FUNCTION_BLOCK Q_ObjHideShow (* Command Hide/Show Object (Container) ( Part 6 - F.2 ) *)
  (* Standard: ISO 11783-6; Description: This command is used to change the value of an object. It applies only to objects that have a numeric value attribute. \retval      iso_s16 - #E_NO_ERR          - OK - #E_OVERFLOW        - buffer overflow - #E_NOACT           - Command not possible in current state - #E_NO_INSTANCE     - No VT client available *)
  (* Version 1.0, 2022-07-08, franz *)
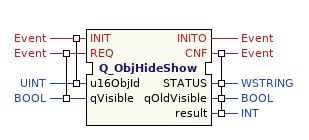
  EVENT_INPUT
    INIT WITH u16ObjId; (* Service Initialization *)
    REQ WITH qVisible; (* Service Request *)
  END_EVENT
  EVENT_OUTPUT
    INITO; (* Initialization Confirm *)
    CNF WITH STATUS, qOldVisible, result; (* Confirmation of Requested Service *)
  END_EVENT
  VAR_INPUT
    u16ObjId : UINT; (* Object ID *)
    qVisible : BOOL; (* 0 == disable, 1 == enable *)
  END_VAR
  VAR_OUTPUT
    STATUS : WSTRING; (* Service Status *)
    qOldVisible : BOOL; (* Old value of Visible *)
    result : INT; (* retval see description *)
  END_VAR
END_FUNCTION_BLOCK
